FUNCTION_BLOCK FB_Stacker EXTENDS FB_Object IMPLEMENTS I_Device

VAR
	nParentSlotNr		: UINT;		//Stacker befindet sich zwar an keinem Slot, aber virtuell in der GUI (am Root)#
	eCurrentState		: E_MachineState := E_MachineState.MACHINESTATE_Idle;
	nNotifyId			: UINT;
	nErrorId			: ERRORID;
	bCanceled			: BOOL;
	bStopAllOnError		: BOOL;
	bIsInit				: BOOL;
	bBusy				: BOOL;
	bError				: BOOL;
	stError				: ST_Error :=(POU := E_POU.POU_FB_Stacker);
	
	nNumberOfShelves	: USINT;
	aShelfes			: ARRAY[1..cMaxShelfes] OF ST_Shelf;
	
	//Hardware-Referenzen
	pHwRef_SpinDrive	: POINTER TO FB_HwRefEL70xxDrive;
	pHwRef_LiftDrive	: POINTER TO FB_HwRefEL70xxDrive;
	pHwRef_TrayStop		: POINTER TO FB_HwRefEL70xxDrive;
	
	bSensorTransAreaLeft 		AT %I* : BOOL;
	bSensorTransAreaRight		AT %I* : BOOL;
	bSensorTrayAlignmentLeft 	AT %I* : BOOL;
	bSensorTrayAlignmentRight 	AT %I* : BOOL;
	bSensorTrayDetection		AT %I* : BOOL;
	
	//Spec-Properties
	nLoadingPosAngle		: DINT;	//Drehwinkel Beladeposition
	nTransferPosAnglePrint1 : DINT;	//Drehwinkel Transferpostion zu Drucker 1
	nTransferPosAnglePrint2 : DINT;	//Drehwinkel Transferpostion zu Drucker 2 (wird derzeit nicht verwendet)
		
	//****************************************Aktionvariablen****************************************************
	
	//Action: "Init"
	bInit				: BOOL;
	nStateA_Init		: USINT;
	fbPower 			: FB_HWECtrl_EL70xx_Power;
	fbHoming 			: FB_HWECtrl_EL70xx_Home;
	pCurrentInitDrive	: POINTER TO FB_HwRefEL70xxDrive;
	
	//Action: "TurnTo"
	bTurnTo				: BOOL;
	nStateA_TurnTo		: USINT;
	fbHwCtrl_Turn		: FB_HWECtrl_EL70xx_Move;
	nTurnToPosition		: DINT;
	
	//Action: "MoveLifter"
	bMoveLifter			: BOOL;
	nStateA_MoveLifter	: USINT;
	nMoveLifterPosition	: DINT;
	nMoveLifterSpeed	: DINT;
	fbHWECtrl_MoveLifter: FB_HWECtrl_EL70xx_Move;
	
	//Action: "OpenCloseTrayStop"
	bOpClTrayStop			: BOOL;
	nStateA_OpClTrayStop	: USINT;
	eOpClTrayStopCtrl		: E_OpClCtrl;
	fbHwCtrl_MoveTrayStop 	: FB_HWECtrl_EL70xx_Move;
	
	//Action: "Load" (Bestücken oder Entnehmen)
	bLoad			: BOOL;
	nStateA_Load	: USINT;
	nBottomShelf	: UINT; //unterstes Fach
	
	stProcessData		: ST_ObjectProcData;
	
END_VAR

VAR CONSTANT
	cMaxShelfes : UINT := 10;
END_VAR

CASE eCurrentState OF
	E_MachineState.MACHINESTATE_Active:
	
		IF bInit THEN
			A_Init();
			IF nStateA_Init >= 80 THEN
				IF nStateA_Init >= 99 THEN
					bError := TRUE;	
				END_IF
				bInit := FALSE;
				nStateA_Init := 0;
			END_IF
		END_IF
		
		IF bTurnTo THEN
			A_TurnTo();
			IF nStateA_TurnTo >= 80 THEN
				IF nStateA_TurnTo >= 99 THEN
					bError := TRUE;	
				END_IF
				bTurnTo := FALSE;
				nStateA_TurnTo := 0;
			END_IF
		END_IF
		
		IF bMoveLifter THEN
			A_MoveLifter();
			IF nStateA_MoveLifter >= 80 THEN
				IF nStateA_MoveLifter >= 99 THEN
					bError := TRUE;	
				END_IF
				bMoveLifter := FALSE;
				nStateA_MoveLifter := 0;
			END_IF
		END_IF
		
		IF bOpClTrayStop THEN
			A_OpClTrayStop();
			IF nStateA_OpClTrayStop >= 80 THEN
				IF nStateA_OpClTrayStop >= 99 THEN
					bError := TRUE;	
				END_IF
				bOpClTrayStop := FALSE;
				nStateA_OpClTrayStop := 0;
			END_IF
		END_IF
		
		IF bLoad THEN
			A_Load();
			IF nStateA_Load >= 80 THEN
				IF nStateA_Load >= 99 THEN
					bError := TRUE;	
				END_IF
				bLoad := FALSE;
				nStateA_Load := 0;
			END_IF
		END_IF
		
		IF NOT (bInit OR bTurnTo OR bMoveLifter OR bOpClTrayStop OR bLoad) THEN
			bBusy := FALSE;
			eCurrentState := E_MachineState.MACHINESTATE_Idle;
		END_IF

		IF bError  THEN
			eCurrentState := E_MachineState.MACHINESTATE_Error;
		END_IF

	E_MachineState.MACHINESTATE_Reset:
		nStateA_Init := 0;
		nStateA_TurnTo := 0;
		nStateA_MoveLifter := 0;
		nStateA_OpClTrayStop := 0;
		nStateA_Load := 0;
		bBusy := FALSE;
		bError := FALSE;
		bStopAllOnError := FALSE;
		stError.Cmd := 0;
		stError.ErrorId := 0;
		eCurrentState := E_MachineState.MACHINESTATE_Idle;
	
	E_MachineState.MACHINESTATE_Error:
		bBusy := FALSE;
END_CASE

//Prozessdaten aktualisieren
stProcessData.nObjId := nObjectID;
stProcessData.n32Data[0] := BOOL_TO_DINT(P_bIsInit);
stProcessData.n32Data[1] := eCurrentState;
stProcessData.n32Data[2] := stError.ErrorId;
stProcessData.n32Data[3] := pHwRef_LiftDrive^.P_nActualPosition;
stProcessData.n32Data[4] := pHwRef_SpinDrive^.P_nActualPosition;
IF pHwRef_TrayStop^.bInput1 THEN //Open
	stProcessData.n32Data[5] := E_OpClState.Open;
ELSIF pHwRef_TrayStop^.bInput2 THEN //Closed
	stProcessData.n32Data[5] := E_OpClState.Closed;
ELSE
	stProcessData.n32Data[5] := E_OpClState.UNDEFINED;
END_IF
	stProcessData.n32Data[6] := BOOL_TO_DINT(bSensorTrayAlignmentLeft AND bSensorTrayAlignmentRight);

aObjProcData[nNotifyId] := stProcessData;

ACTION A_Init:
stError.POUState := nStateA_Init;

CASE nStateA_Init OF
	0:	//Power TrayStop
		pCurrentInitDrive := pHwRef_TrayStop;
		fbPower(pHwRef:= pHwRef_TrayStop, bEnable:= TRUE, bExecute:= TRUE);
		IF NOT fbPower.bBusy THEN
			IF fbPower.bError THEN
				stError.ErrorId := fbPower.nErrorId;
				nStateA_Init := 99;
			ELSE
				nStateA_Init := 1;
			END_IF
			fbPower(pHwRef := pHwRef_TrayStop, bExecute:= FALSE);
		END_IF
		
	1:	//Power SpinDrive
		pCurrentInitDrive := pHwRef_SpinDrive;
		fbPower(pHwRef:= pHwRef_SpinDrive, bEnable:= TRUE, bExecute:= TRUE);
		IF NOT fbPower.bBusy THEN
			IF fbPower.bError THEN
				stError.ErrorId := fbPower.nErrorId;
				nStateA_Init := 99;
			ELSE
				nStateA_Init := 2;
			END_IF
			fbPower(pHwRef:= pHwRef_SpinDrive, bExecute:= FALSE);
		END_IF

	2:	//Power LiftDrive
		pCurrentInitDrive := pHwRef_LiftDrive;
		fbPower(pHwRef:= pHwRef_LiftDrive, bEnable:= TRUE, bExecute:= TRUE);
		IF NOT fbPower.bBusy THEN
			IF fbPower.bError THEN
				stError.ErrorId := fbPower.nErrorId;
				nStateA_Init := 99;
			ELSE
				nStateA_Init := 3;
			END_IF
			fbPower(pHwRef:= pHwRef_LiftDrive, bExecute:= FALSE);
		END_IF
		
	3:	//Homing TrayStop
		pCurrentInitDrive := pHwRef_TrayStop;
		fbHoming(pHwRef:= pHwRef_TrayStop, bExecute:= TRUE);
		IF NOT fbHoming.bBusy THEN
			IF fbHoming.bError THEN
				stError.ErrorId := fbHoming.nErrorId;
				nStateA_Init := 99;
			ELSE
				nStateA_Init := 4;
			END_IF
			fbHoming(pHwRef:= pHwRef_TrayStop, bExecute:= FALSE);
		END_IF

	4:	//Homing SpinDrive
		pCurrentInitDrive := pHwRef_SpinDrive;
		fbHoming(pHwRef:= pHwRef_SpinDrive, bExecute:= TRUE);
		IF NOT fbHoming.bBusy THEN
			IF fbHoming.bError THEN
				stError.ErrorId := fbHoming.nErrorId;
				nStateA_Init := 99;
			ELSE
				nStateA_Init := 5;
			END_IF
			fbHoming(pHwRef:= pHwRef_SpinDrive, bExecute:= FALSE);
		END_IF
		
	5:	//Homing LiftDrive
		pCurrentInitDrive := pHwRef_LiftDrive;
		//TransArea überwachen
		IF NOT P_bTransAreaFree THEN
			//Stoppen und dann in Error
			fbHoming(pHwRef:= pHwRef_LiftDrive, bStop := TRUE);
			nStateA_Init := 75;
		ELSE
			fbHoming(pHwRef:= pHwRef_LiftDrive, bExecute:= TRUE);
			IF NOT fbHoming.bBusy THEN
				IF fbHoming.bError THEN
					stError.ErrorId := fbHoming.nErrorId;
					nStateA_Init := 99;
				ELSE
					nStateA_Init := 80;
				END_IF
				fbHoming(pHwRef:= pHwRef_LiftDrive, bExecute:= FALSE);
			END_IF
		END_IF
		
	70:	//Abbrechen
		IF fbPower.bBusy THEN //Warten bis fbPower fertig
			nStateA_Init := 71;
		ELSIF fbHoming.bBusy THEN
			nStateA_Init := 72;
		ELSE
			nStateA_Init := 80;
		END_IF
		
	71:	//Power ready?
		fbPower(pHwRef:= pCurrentInitDrive);
		IF NOT fbPower.bBusy THEN
			fbPower(pHwRef:= pCurrentInitDrive, bExecute := FALSE);
			nStateA_Init := 80;
		END_IF
		
	72:	//Homing abbrechen
		fbHoming(pHwRef:= pCurrentInitDrive, bStop:= TRUE);
		IF NOT fbHoming.bBusy THEN
			fbHoming(pHwRef:= pCurrentInitDrive, bStop:= FALSE, bExecute := FALSE);
			nStateA_Init := 80;
		END_IF
		
	75:	//Homing Lifter abbrechen und dann in Error
		fbHoming(pHwRef:= pCurrentInitDrive, bStop:= TRUE);
		IF NOT fbHoming.bBusy THEN
			fbHoming(pHwRef:= pCurrentInitDrive, bStop:= FALSE, bExecute := FALSE);
			stError.ErrorId := E_ErrorIdCmd.ERRORID_TransferAreaNotFree;
			nStateA_Init := 99;
		END_IF
 	
END_CASE

//Errorhandling
IF nStateA_Init = 99 THEN
	stError.ObjectId := nObjectID;
	stError.Cmd := E_Action.ACTION_Init;
	stError.POUAction := E_POUACT.POUACT_A_Init;
	fbErrorList.M_Add(stError);
END_IF
END_ACTION

ACTION A_Load:
//Diese Action darf nur ausgeführt werden, wenn:
//Initialisiert ist
//keine andere Action aktiv ist
//Es werden alle Actions einzeln ausgeführt.
//1. turn
//2. move lifter
//3. close tray stopper
//4. open interlock

CASE nStateA_Load OF
	0:	//Turn to loading position
		nTurnToPosition := nLoadingPosAngle;
		A_TurnTo();
		IF nStateA_TurnTo >= 80 THEN
			IF nStateA_TurnTo >= 99 THEN
				nStateA_Load := 99;
			ELSE
				nStateA_Load := 1;
			END_IF
			nStateA_TurnTo := 0;
		END_IF

	1:	//Move lifter
		nMoveLifterPosition := M_GetBottomShelfPos();
		nMoveLifterSpeed := pHwRef_LiftDrive^.P_nMaxSpeed;
		A_MoveLifter();
		IF nStateA_MoveLifter >= 80 THEN
			IF nStateA_MoveLifter >= 99 THEN
				nStateA_Load := 99;
			ELSE
				nStateA_Load := 2;
			END_IF
			nStateA_MoveLifter := 0;
		END_IF
				
	2:	//Close tray stopper
		eOpClTrayStopCtrl := E_OpClCtrl.Close;
		A_OpClTrayStop();
		IF nStateA_OpClTrayStop >= 80 THEN
			IF nStateA_OpClTrayStop >= 99 THEN
				nStateA_Load := 99;
			ELSE
				nStateA_Load := 3;
			END_IF
			nStateA_OpClTrayStop := 0;
		END_IF
		
	3:	//Open interlock stacker
		{IF defined(Stacker)}
		fbSafetyStacker.M_Control(E_SafetyCtrl.Unlock);
		{END_IF}
		nStateA_Load := 80;
	
	70:	//Cancel
		//Which actin is active?
		//we can identify the active action wich nStateA_xxxx is greather than 0
		IF nStateA_TurnTo > 0 THEN
			;
		ELSIF nStateA_MoveLifter > 0 THEN
			;
		ELSIF nStateA_OpClTrayStop > 0 THEN
			;
		END_IF
	
	
END_CASE
END_ACTION

ACTION A_MoveLifter:
IF nStateA_MoveLifter = 0 THEN
	//Nur TransArea überwachen	
	IF NOT P_bTransAreaFree THEN
		//Stoppen und dann in Error
		fbHWECtrl_MoveLifter(pHwRef:= pHwRef_LiftDrive, bStop:= TRUE);
		nStateA_MoveLifter := 75;
	ELSE
		fbHWECtrl_MoveLifter(pHwRef:= pHwRef_LiftDrive, nPosition := nMoveLifterPosition, nSpeed:= nMoveLifterSpeed, bExecute:= TRUE);
		IF NOT fbHWECtrl_MoveLifter.bBusy THEN
			IF fbHWECtrl_MoveLifter.bError THEN
				stError.ErrorId := fbHWECtrl_MoveLifter.nErrorId;
				nStateA_MoveLifter := 99;
			ELSE
				nStateA_MoveLifter := 80;
			END_IF
			fbHWECtrl_MoveLifter(pHwRef:= pHwRef_LiftDrive, bExecute:= FALSE);
		END_IF
	END_IF
	
ELSIF nStateA_MoveLifter = 70 THEN //Normal stoppen
	fbHWECtrl_MoveLifter(pHwRef:= pHwRef_LiftDrive, bStop := TRUE);
	IF NOT fbHWECtrl_MoveLifter.bBusy THEN
		IF fbHWECtrl_MoveLifter.bError THEN
			stError.ErrorId := fbHWECtrl_MoveLifter.nErrorId;
			nStateA_MoveLifter := 99;
		ELSE
			nStateA_MoveLifter := 80;
		END_IF
		fbHWECtrl_MoveLifter(pHwRef:= pHwRef_LiftDrive, bExecute:= FALSE);
	END_IF
	
ELSIF nStateA_MoveLifter = 75 THEN //Stoppen mit folgender Error-Meldung
	fbHWECtrl_MoveLifter(pHwRef:= pHwRef_LiftDrive);
	IF NOT fbHWECtrl_MoveLifter.bBusy THEN
		IF fbHWECtrl_MoveLifter.bError THEN
			stError.ErrorId := fbHWECtrl_MoveLifter.nErrorId;
		ELSE
			stError.ErrorId := E_ErrorIdCmd.ERRORID_TransferAreaNotFree;
		END_IF
		fbHWECtrl_MoveLifter(pHwRef:= pHwRef_LiftDrive, bExecute:= FALSE);
		nStateA_MoveLifter := 99;
	END_IF
END_IF

//Errorhandling
IF nStateA_MoveLifter = 99 THEN
	stError.ObjectId := nObjectID;
	stError.Cmd := E_Action.ACTION_MoveLifter;
	stError.POUAction := E_POUACT.POUACT_A_MoveLifter;
	fbErrorList.M_Add(stError);
END_IF
END_ACTION

ACTION A_OpClTrayStop:
IF nStateA_OpClTrayStop = 0 THEN
	IF eOpClTrayStopCtrl = E_OpClCtrl.Close THEN
		fbHwCtrl_MoveTrayStop(pHwRef:= pHwRef_TrayStop, nPosition:= pHwRef_TrayStop^.P_nMaxPos, nSpeed:= pHwRef_TrayStop^.P_nMaxSpeed, bExecute:= TRUE);
		nStateA_OpClTrayStop := 1;
	ELSE
		fbHwCtrl_MoveTrayStop(pHwRef:= pHwRef_TrayStop, nPosition:= 0, nSpeed:= pHwRef_TrayStop^.P_nMaxSpeed, bExecute:= TRUE);
		nStateA_OpClTrayStop := 1;
	END_IF
ELSIF nStateA_OpClTrayStop = 1 THEN
	fbHwCtrl_MoveTrayStop(pHwRef:= pHwRef_TrayStop);
	IF NOT fbHwCtrl_MoveTrayStop.bBusy THEN
		IF fbHwCtrl_MoveTrayStop.bError THEN
			stError.ErrorId := fbHwCtrl_MoveTrayStop.nErrorId;
			nStateA_OpClTrayStop := 99;
		ELSE
			IF eOpClTrayStopCtrl = E_OpClCtrl.Close THEN
				IF pHwRef_TrayStop^.bInput2 THEN
					nStateA_OpClTrayStop := 80;
				ELSE
					stError.ErrorId := E_ErrorIdCmd.ERRORID_TrayStopNotClosed;
					nStateA_OpClTrayStop := 99;
				END_IF
			ELSE
				IF pHwRef_TrayStop^.bInput1 THEN
					nStateA_OpClTrayStop := 80;
				ELSE
					stError.ErrorId := E_ErrorIdCmd.ERRORID_TrayStopNotOpen;
					nStateA_OpClTrayStop := 99;
				END_IF
			END_IF
		END_IF
		fbHwCtrl_MoveTrayStop(pHwRef:= pHwRef_TrayStop, bExecute:= FALSE);
	END_IF
ELSIF nStateA_OpClTrayStop = 70 THEN
	fbHwCtrl_MoveTrayStop(pHwRef:= pHwRef_TrayStop, bStop := TRUE);
	IF NOT fbHwCtrl_MoveTrayStop.bBusy THEN
		IF fbHwCtrl_MoveTrayStop.bError THEN
			stError.ErrorId := fbHwCtrl_MoveTrayStop.nErrorId;
			nStateA_OpClTrayStop := 99;
		ELSE
			nStateA_OpClTrayStop := 80;
		END_IF
		fbHwCtrl_MoveTrayStop(pHwRef:= pHwRef_TrayStop, bExecute:= FALSE);
	END_IF
	
END_IF

//Errorhandling
IF nStateA_OpClTrayStop = 99 THEN
	stError.ObjectId := nObjectID;
	stError.Cmd := E_Action.ACTION_OpenClose;
	stError.POUAction := E_POUACT.POUACT_A_OpClTrayStop;
	fbErrorList.M_Add(stError);
END_IF
END_ACTION

ACTION A_TurnTo:
IF nStateA_TurnTo = 0 THEN
	fbHwCtrl_Turn(pHwRef:= pHwRef_SpinDrive, nPosition:= nTurnToPosition, nSpeed:= pHwRef_SpinDrive^.P_nMaxSpeed,
					nToleranceWindow:= 50, bExecute:= TRUE);
	IF NOT fbHwCtrl_Turn.bBusy THEN
		IF fbHwCtrl_Turn.bError THEN
			stError.ErrorId := fbHwCtrl_Turn.nErrorId;
			nStateA_TurnTo := 99;
		ELSE
			nStateA_TurnTo := 80;
		END_IF
		fbHwCtrl_Turn(pHwRef:= pHwRef_SpinDrive, bExecute := FALSE);
	END_IF
ELSIF nStateA_TurnTo = 70 THEN
	fbHwCtrl_Turn(pHwRef:= pHwRef_SpinDrive, bStop:= TRUE);
	IF NOT fbHwCtrl_Turn.bBusy THEN
		IF fbHwCtrl_Turn.bError THEN
			stError.ErrorId := fbHwCtrl_Turn.nErrorId;
			nStateA_TurnTo := 99;
		ELSE
			nStateA_TurnTo := 80;
		END_IF
		fbHwCtrl_Turn(pHwRef:= pHwRef_SpinDrive, bExecute := FALSE);
	END_IF	
END_IF

//Errorhandling
IF nStateA_TurnTo = 99 THEN
	stError.ObjectId := nObjectID;
	stError.Cmd := E_Action.ACTION_TurnTo;
	stError.POUAction := E_POUACT.POUACT_A_TurnTo;
	fbErrorList.M_Add(stError);
END_IF
END_ACTION

METHOD FB_init : BOOL
VAR_INPUT
	bInitRetains 		: BOOL; // if TRUE, the retain variables are initialized (warm start / cold start)
	bInCopyCode 		: BOOL;  // if TRUE, the instance afterwards gets moved into the copy code (online change)
END_VAR
eObjectType := E_ObjectType.OBJECTTYPE_Stacker;
eObjectGroup := E_ObjectGroup.OBJECTGROUP_Device;
END_METHOD

METHOD M_CancelAction
VAR_INPUT
	eAction : E_Action;
END_VAR
CASE eAction OF
	E_Action.ACTION_Init:
		IF bInit AND nStateA_Init < 70 THEN
			nStateA_Init := 70;
		END_IF
		
	E_Action.ACTION_TurnTo:
		IF bTurnTo AND nStateA_TurnTo < 70 THEN
			nStateA_TurnTo := 70;
		END_IF
		
	E_Action.ACTION_MoveLifter:
		IF bMoveLifter AND nStateA_MoveLifter < 70 THEN
			nStateA_MoveLifter := 70;
		END_IF
		
	E_Action.ACTION_OpenClose:
		IF bOpClTrayStop AND nStateA_OpClTrayStop < 70 THEN
			nStateA_OpClTrayStop := 70;
		END_IF
		
END_CASE
END_METHOD

METHOD M_CheckAction : ERRORID
VAR_INPUT
	refActionData 	: REFERENCE TO ST_ActionData;
	pCorrelObject	: POINTER TO FB_Object;
END_VAR
M_CheckAction := E_ErrorIdCmd.ERRORID_InvalidAction;
END_METHOD

METHOD M_CheckProcDataType : BOOL
VAR_INPUT
	eProcDataType : E_ProcDataType;
END_VAR
END_METHOD

METHOD M_ClearAllProps
VAR_INPUT
	bIgnoreParent : BOOL; //Es wird das gesamte OD gelöscht. -> Zeiger auf Parent nicht mehr gültig!	
END_VAR
MEMSET(ADR(aShelfes), 0, SIZEOF(aShelfes));
END_METHOD

METHOD M_ExeAction : ERRORID
VAR_INPUT
	refActionData	: REFERENCE TO ST_ActionData;
END_VAR


VAR
	eStackerRotPosition : E_StackerRotPosition;
END_VAR
//Stacker ist so implementiet, dass mehrere Actions nicht zeitgleich ausgeführt werden können.
//Das bedeutet, dass eCurrentState idle sein muss
IF eCurrentState = E_MachineState.MACHINESTATE_Active THEN
	M_ExeAction := E_ErrorIdCmd.ERRORID_BasicActionActive;
	RETURN;	
ELSIF eCurrentState = E_MachineState.MACHINESTATE_Error OR eCurrentState = E_MachineState.MACHINESTATE_Reset THEN
	M_ExeAction := E_ErrorIdCmd.ERRORID_InvalidState;
	RETURN;	
END_IF

IF refActionData.eAction <> E_Action.ACTION_Init THEN
	IF NOT P_bIsInit THEN
		M_ExeAction := E_ErrorIdCmd.ERRORID_DeviceNotInitialized;
		RETURN;
	END_IF
END_IF

{IF defined(Stacker)}
IF fbSafetyStacker.eCurrentState <> E_SafetyState.Locked THEN
	M_ExeAction := E_ErrorIdCmd.ERRORID_InterlockNotLocked;
END_IF
{END_IF}

CASE refActionData.eAction OF
	E_Action.ACTION_Init:
		IF NOT bInit THEN
			IF NOT P_bTransAreaFree THEN
				M_ExeAction := E_ErrorIdCmd.ERRORID_TransferAreaNotFree;
				RETURN;
			END_IF
			
			IF NOT P_bTraysAligned THEN
				M_ExeAction := E_ErrorIdCmd.ERRORID_TraysNotAligned;
				RETURN;
			END_IF
			bInit := TRUE;
		ELSE
			RETURN;
		END_IF

	E_Action.ACTION_TurnTo:
		IF NOT bTurnTo THEN
			IF NOT P_bTransAreaFree THEN
				M_ExeAction := E_ErrorIdCmd.ERRORID_TransferAreaNotFree;
				RETURN;
			END_IF
			
			IF NOT P_bTraysAligned THEN
				M_ExeAction := E_ErrorIdCmd.ERRORID_TraysNotAligned;
				RETURN;
			END_IF
			
			eStackerRotPosition := DINT_TO_USINT(refActionData.aParams[1]);
			CASE eStackerRotPosition OF
				E_StackerRotPosition.LoadingPosition:
					nTurnToPosition := nLoadingPosAngle;
				E_StackerRotPosition.TransferPositionPrinter1:
					nTurnToPosition := nTransferPosAnglePrint1;
				E_StackerRotPosition.TransferPositionPrinter2:
					nTurnToPosition := nTransferPosAnglePrint2;
			ELSE
				M_ExeAction := E_ErrorIdCmd.ERRORID_InvalidStackerAngle;
				RETURN;
			END_CASE
			bTurnTo := TRUE;
		ELSE
			RETURN;
		END_IF
		
	E_Action.ACTION_MoveLifter:
		IF NOT bMoveLifter THEN
			IF NOT P_bTransAreaFree THEN
				M_ExeAction := E_ErrorIdCmd.ERRORID_TransferAreaNotFree;
				RETURN;
			END_IF
			
			IF NOT P_bTraysAligned THEN
				M_ExeAction := E_ErrorIdCmd.ERRORID_TraysNotAligned;
				RETURN;
			END_IF
			
			nMoveLifterPosition := refActionData.aParams[1];
			nMoveLifterSpeed := refActionData.aParams[2];
			bMoveLifter := TRUE;
		ELSE
			RETURN;
		END_IF
		
	E_Action.ACTION_OpenClose:
		IF NOT bOpClTrayStop THEN
			eOpClTrayStopCtrl := DINT_TO_USINT(refActionData.aParams[1]);
			bOpClTrayStop := TRUE;
		ELSE
			RETURN;
		END_IF
		
	E_Action.ACTION_LoadStacker:
		IF NOT P_bTransAreaFree THEN
			M_ExeAction := E_ErrorIdCmd.ERRORID_TransferAreaNotFree;
			RETURN;
		END_IF
		
		IF NOT P_bTraysAligned THEN
			M_ExeAction := E_ErrorIdCmd.ERRORID_TraysNotAligned;
			RETURN;
		END_IF
		
		IF NOT bLoad THEN
			bLoad := TRUE;
		ELSE
			RETURN;
		END_IF
	
END_CASE

eCurrentState := E_MachineState.MACHINESTATE_Active;
bBusy := TRUE;
END_METHOD

METHOD M_GetActionBusy : BOOL
VAR_INPUT
	eAction : E_Action;
END_VAR
CASE eAction OF
	E_Action.ACTION_Init:
		M_GetActionBusy := bInit;
	E_Action.ACTION_TurnTo:
		M_GetActionBusy := bTurnTo;
	E_Action.ACTION_MoveLifter:
		M_GetActionBusy := bMoveLifter;
	E_Action.ACTION_OpenClose:
		M_GetActionBusy := bOpClTrayStop;
	E_Action.ACTION_LoadStacker:
		M_GetActionBusy := bLoad;
END_CASE
END_METHOD

METHOD M_GetAllProps : ERRORID
VAR_INPUT
	refCmdData : REFERENCE TO  ST_CmdData;
END_VAR

VAR
	nCurrentPropIndex	: UINT;
	i : UINT;
END_VAR
refCmdData.aHeader[0] := nObjectID;
refCmdData.aHeader[1] := eObjectType;
refCmdData.aHeader[2]:= nNotifyId;

nCurrentPropIndex := 1;
refCmdData.n32Data[nCurrentPropIndex] := nParentSlotNr;
nCurrentPropIndex := nCurrentPropIndex + 1;
refCmdData.n32Data[nCurrentPropIndex] := nNumberOfShelves;
FOR i := 1 TO nNumberOfShelves DO
	nCurrentPropIndex := nCurrentPropIndex + 1;
	refCmdData.n32Data[nCurrentPropIndex] := aShelfes[i].nPosition;	
END_FOR
nCurrentPropIndex := nCurrentPropIndex + 1;
refCmdData.n32Data[nCurrentPropIndex] := nLoadingPosAngle;
nCurrentPropIndex := nCurrentPropIndex + 1;
refCmdData.n32Data[nCurrentPropIndex] := nTransferPosAnglePrint1;
nCurrentPropIndex := nCurrentPropIndex + 1;
refCmdData.n32Data[nCurrentPropIndex] := nTransferPosAnglePrint2;
END_METHOD

METHOD M_GetBottomShelfPos : DINT
VAR_INPUT
END_VAR

VAR
	i 		: UINT;
	nPos	: DINT;
END_VAR
FOR i := 1 TO nNumberOfShelves DO
	IF aShelfes[i].nPosition > nPos THEN
		nPos :=	aShelfes[i].nPosition;
	END_IF
END_FOR
M_GetBottomShelfPos := nPos;
END_METHOD

METHOD M_GetDevice : I_Device
VAR_INPUT
END_VAR
M_GetDevice := THIS^;
END_METHOD

METHOD M_GetProcData : DINT
VAR_INPUT
	eProcDataType : E_ProcDataType;
END_VAR
END_METHOD

METHOD M_Reset
bBusy := TRUE;
eCurrentState := E_MachineState.MACHINESTATE_Reset;
END_METHOD

METHOD M_SetAllProps : ERRORID
VAR_INPUT
	refCmdData : REFERENCE TO  ST_CmdData;
END_VAR

VAR
	i : UINT;
	nCurrentPropIndex	: UINT;
END_VAR
nCurrentPropIndex := 1;
nParentSlotNr := DINT_TO_UINT(refCmdData.n32Data[nCurrentPropIndex]);
nCurrentPropIndex := nCurrentPropIndex + 1;
//Shelfes (Fächer) parametrieren
nNumberOfShelves := DINT_TO_USINT(refCmdData.n32Data[nCurrentPropIndex]);
IF nNumberOfShelves > cMaxShelfes THEN
	M_SetAllProps := E_ErrorIdObjMgmt.ERRORID_InvalidNumberOfShelfes;
	RETURN;
END_IF

FOR i := 1 TO nNumberOfShelves DO
	nCurrentPropIndex := nCurrentPropIndex + 1;
	aShelfes[i].nPosition := refCmdData.n32Data[nCurrentPropIndex];
	aShelfes[i].bConfigured := TRUE;
END_FOR

{IF defined (Stacker)}
	pHwRef_SpinDrive := ADR(fbHwRefSpinDrive);
	pHwRef_LiftDrive := ADR(fbHwRefLiftDrive);
	pHwRef_TrayStop := ADR(fbHwRefTrayStop);
{ELSE}
	M_SetAllProps := E_ErrorIdObjMgmt.ERRORID_Stacker_NotDefined;
	RETURN;
{END_IF}

nCurrentPropIndex := nCurrentPropIndex + 1;
nLoadingPosAngle := refCmdData.n32Data[nCurrentPropIndex];
nCurrentPropIndex := nCurrentPropIndex + 1;
nTransferPosAnglePrint1 := refCmdData.n32Data[nCurrentPropIndex];
nCurrentPropIndex := nCurrentPropIndex + 1;
nTransferPosAnglePrint2 := refCmdData.n32Data[nCurrentPropIndex];
nNoOfProps := nCurrentPropIndex + 1;
END_METHOD

METHOD M_SetSingleProp : ERRORID
VAR_INPUT
	refCmdData : REFERENCE TO  ST_CmdData;
END_VAR
(*IF nSpecPropIndex = refCmdData.aHeader[1] THEN
	nLoadingPosAngle := refCmdData.n32Data[0];
ELSIF (nSpecPropIndex + 1) = refCmdData.aHeader[1] THEN
	nTransferPosAnglePrint1 := refCmdData.n32Data[0];
ELSIF (nSpecPropIndex + 2) = refCmdData.aHeader[1] THEN
	nTransferPosAnglePrint2 := refCmdData.n32Data[0];
ELSE
	M_SetSingleProp := SUPER^.M_SetSingleProp(refCmdData);
END_IF*)
END_METHOD

METHOD M_Stop : ERRORID
IF eCurrentState = E_MachineState.MACHINESTATE_Active THEN
	IF bInit AND nStateA_Init < 70 THEN
		nStateA_Init := 70;
	END_IF
	
	IF bTurnTo AND nStateA_TurnTo < 70 THEN
		nStateA_TurnTo := 70;
	END_IF
	
	IF bMoveLifter AND nStateA_MoveLifter < 70 THEN
		nStateA_MoveLifter := 70;
	END_IF
	
	IF bOpClTrayStop AND nStateA_OpClTrayStop < 70 THEN
		nStateA_OpClTrayStop := 70;
	END_IF	
END_IF
END_METHOD

PROPERTY P_bBusy : BOOL
GET
P_bBusy := bBusy;
END_GET
END_PROPERTY

PROPERTY P_bCanceled : BOOL
GET
P_bCanceled := bCanceled;
END_GET
END_PROPERTY

PROPERTY P_bError : BOOL
GET
P_bError := (eCurrentState = E_MachineState.MACHINESTATE_Error);
END_GET
END_PROPERTY

PROPERTY P_bIsInit : BOOL
GET
IF pHwRef_SpinDrive > 0 AND_THEN pHwRef_LiftDrive > 0 AND_THEN pHwRef_TrayStop > 0 THEN
	P_bIsInit := pHwRef_SpinDrive^.P_bIsInit AND pHwRef_LiftDrive^.P_bIsInit AND pHwRef_TrayStop^.P_bIsInit;
END_IF
END_GET
SET
bIsInit := P_bIsInit;
END_SET
END_PROPERTY

PROPERTY P_bStopAllOnError : BOOL
GET
P_bStopAllOnError := bStopAllOnError;
END_GET
END_PROPERTY

PROPERTY P_bTransAreaFree : BOOL
GET
P_bTransAreaFree := TRUE;
IF F_GetMappingStatus(ADR(bSensorTransAreaLeft),SIZEOF(bSensorTransAreaLeft)) = EPlcMappingStatus.MS_Partial THEN
	IF NOT bSensorTransAreaLeft THEN
		P_bTransAreaFree := FALSE;
	END_IF
END_IF

IF F_GetMappingStatus(ADR(bSensorTransAreaRight),SIZEOF(bSensorTransAreaRight)) = EPlcMappingStatus.MS_Partial THEN
	IF NOT bSensorTransAreaRight THEN
		P_bTransAreaFree := FALSE;
	END_IF	
END_IF
END_GET
END_PROPERTY

PROPERTY P_bTrayInCurrentShelf : BOOL
GET
P_bTrayInCurrentShelf := bSensorTrayDetection;
END_GET
END_PROPERTY

PROPERTY P_bTraysAligned : BOOL
GET
P_bTraysAligned := bSensorTrayAlignmentLeft AND bSensorTrayAlignmentRight;
END_GET
END_PROPERTY

PROPERTY P_eCurrentSpinPositon : E_StackerRotPosition
GET
VAR
	nActPosTemp : DINT;
END_VAR
IF pHwRef_SpinDrive^.P_nActualPosition > 359000 THEN
	nActPosTemp := -(360000 - pHwRef_SpinDrive^.P_nActualPosition);
ELSE
	nActPosTemp := pHwRef_SpinDrive^.P_nActualPosition;
END_IF

IF nActPosTemp >= (nLoadingPosAngle - 100) AND nActPosTemp <= (nLoadingPosAngle + 100) THEN
	P_eCurrentSpinPositon := E_StackerRotPosition.LoadingPosition;
ELSIF nActPosTemp >= (nTransferPosAnglePrint1 - 100) AND nActPosTemp <= (nTransferPosAnglePrint1 + 100) THEN
	P_eCurrentSpinPositon := E_StackerRotPosition.TransferPositionPrinter1;
ELSIF nActPosTemp >= (nTransferPosAnglePrint2 - 100) AND nActPosTemp <= (nTransferPosAnglePrint2 + 100) THEN
	P_eCurrentSpinPositon := E_StackerRotPosition.TransferPositionPrinter2;
ELSE
	P_eCurrentSpinPositon := E_StackerRotPosition.UNDEFINED;
END_IF
END_GET
END_PROPERTY

PROPERTY P_eCurrentState : E_MachineState
GET
P_eCurrentState := eCurrentState;
END_GET
END_PROPERTY

PROPERTY P_nCurrentShelf : UINT
GET
VAR
	i : USINT;
END_VAR
FOR i := 1 TO nNumberOfShelves DO
	IF pHwRef_LiftDrive^.P_nActualPosition >= aShelfes[i].nPosition - 200 AND pHwRef_LiftDrive^.P_nActualPosition <= aShelfes[i].nPosition + 200 THEN
		P_nCurrentShelf := i;
		EXIT;
	END_IF
END_FOR
END_GET
END_PROPERTY

PROPERTY P_nErrorId : ERRORID
GET
P_nErrorID := stError.ErrorId;
END_GET
END_PROPERTY

PROPERTY P_nNotifyId : UINT
GET
P_nNotifyId := nNotifyId;
END_GET
SET
nNotifyId := P_nNotifyId;
END_SET
END_PROPERTY

PROPERTY P_nParentSlotNr : UINT
GET
P_nParentSlotNr := nParentSlotNr;
END_GET
END_PROPERTY

PROPERTY P_pObject : POINTER TO FB_Object
GET
P_pObject := THIS;
END_GET
END_PROPERTY

PROPERTY P_stError : ST_Error
GET
END_GET
END_PROPERTY

END_FUNCTION_BLOCK

(* stored: Version 1.1.0.1, ProductVersion 3.1.4024.11
   POU FB_Stacker: Id {f8d592f7-3fdb-4527-8cd4-2934179103ba}, SpecialFunc None
   Action A_Init: Id {6a4671f8-a2b8-4336-b86c-03d30b71aca8}
   Action A_Load: Id {e778a475-0736-4db9-b8d8-85e9b4b33938}
   Action A_MoveLifter: Id {bdc9ef98-55ce-4c64-b557-b10613fc331f}
   Action A_OpClTrayStop: Id {fad61029-ac97-4061-82b7-aa3f29a40dba}
   Action A_TurnTo: Id {236ce99b-081e-458c-8081-62ddfff656f2}
   Method FB_init: Id {f9a7eb7f-9be7-4bc9-953c-9146258cbf9c}
   Method M_CancelAction: Id {52aeec01-1bfb-4d1e-a15b-ca58b70141c6}
   Method M_CheckAction: Id {cdd695e1-2576-4bf3-aeea-155881d07d0c}
   Method M_CheckProcDataType: Id {097f035e-a523-4887-a70f-c028028da1da}
   Method M_ClearAllProps: Id {766e1508-7eb0-4d9d-b34f-fa0031c4612d}
   Method M_ExeAction: Id {c158a3da-a343-4259-b179-02467dfff6a8}
   Method M_GetActionBusy: Id {4456857c-8d47-4244-b2f0-54a996bd0baa}
   Method M_GetAllProps: Id {98ef0bf2-59e0-4987-aa75-3f69b4ec7e59}
   Method M_GetBottomShelfPos: Id {337386ba-3fa1-4591-946b-350815013f06}
   Method M_GetDevice: Id {d246706d-af2e-4004-88c5-f7b70cc1781a}
   Method M_GetProcData: Id {32a87474-f5b7-4b4b-9af0-13cfd7ee5835}
   Method M_Reset: Id {1020664e-004e-41e5-897d-2290e44b8ebe}
   Method M_SetAllProps: Id {a7e0c6d5-8999-4f49-8640-388d6dd9fbff}
   Method M_SetSingleProp: Id {d842e7bc-c393-4c16-beba-31952210c5cb}
   Method M_Stop: Id {1ad0d9cd-a1b7-4420-a794-812f186f2be3}
   Property P_bBusy: Id {71b7153d-014e-4044-8913-fdce658a022e}
   Get Get: Id {d86098cb-740c-4d42-867f-6e2825ebc35b}
   Property P_bCanceled: Id {f96a21d4-c8a5-4077-8e97-2bb648a3a493}
   Get Get: Id {116a37a3-45f0-49c8-885c-19aeeb74dd55}
   Property P_bError: Id {7ec15977-d0db-4829-b35b-c8087c2b92a9}
   Get Get: Id {7f867612-b7c4-4824-ad64-08649b2d4a1b}
   Property P_bIsInit: Id {ac53ed0f-659a-4975-951e-71afcec80129}
   Get Get: Id {935d605e-c41a-4a30-be0d-dd482a8b0a19}
   Set Set: Id {6484b4fe-912a-4d05-808b-88275c5d7690}
   Property P_bStopAllOnError: Id {77900df0-4a56-49c8-9b32-df76e299fb94}
   Get Get: Id {37d64613-7882-4ac4-9d9d-f55fad5965e6}
   Property P_bTransAreaFree: Id {e38fb50b-44c8-440e-8214-b2b569b51375}
   Get Get: Id {a8af8630-d44c-4f87-b5de-f190505aefcc}
   Property P_bTrayInCurrentShelf: Id {69a22060-8837-423f-b5f8-200b6238ffd2}
   Get Get: Id {60fff5b7-61cd-469a-af9a-ae8ff34d66c5}
   Property P_bTraysAligned: Id {a8828430-b492-4142-9d65-b89bfb6b62e1}
   Get Get: Id {c1a2c6cb-f0fa-4848-b02a-e83d0b2d1fea}
   Property P_eCurrentSpinPositon: Id {3206e673-f0f5-4bd7-9945-06da70f5b2c6}
   Get Get: Id {1d04ee20-06da-4582-a47e-e5b9842e8bb0}
   Property P_eCurrentState: Id {e23c968c-9a73-4198-b0ff-88105f5ba9b2}
   Get Get: Id {d56ba0af-dc92-43f1-b47f-9b63d86b6b62}
   Property P_nCurrentShelf: Id {1f0642f9-267f-42d5-9605-9f1ed3d48939}
   Get Get: Id {2e8f0b79-d584-46ab-b308-7a7339c1edcb}
   Property P_nErrorId: Id {26cff18c-7749-472f-bb8e-c0af379b4018}
   Get Get: Id {b9c50be7-3808-4ac2-ae99-c81712fb1cff}
   Property P_nNotifyId: Id {b562c9f4-924a-430d-8bd3-1737e4dde26e}
   Get Get: Id {de32249a-85de-4af9-8438-f96899e75415}
   Set Set: Id {fb1393aa-5627-49e8-8f87-e3f7b7a90c7e}
   Property P_nParentSlotNr: Id {8271ac5e-5983-4a97-bb85-ec242f0a92b3}
   Get Get: Id {49c0bf64-c1bf-4bb3-9310-794285aa8083}
   Property P_pObject: Id {a2af1854-1d68-49fc-9cd7-29dcaebb1481}
   Get Get: Id {d3b9cd7e-b019-4a6c-a035-5028903f2ae0}
   Property P_stError: Id {ff000683-0cf0-4426-aad0-249928972c9c}
   Get Get: Id {e0d85a98-4653-4d37-84cb-d97bcdd426f8} *)
